(* IEC 61131-3 sources: 2026_Projet_YGO_ExcavatriceDragage/TOOLS/TEST_AUTO_CI/RESULTS/MAIN, 5 files *)

(* ---- FB_Main_EndToEnd.st ---- *)
(* =======================================================================
   🏰 FB_Main_EndToEnd : Mégabloc Machine d'Intégration Globale
   ───────────────────────────────────────────────────────────────
   🎯 Rôle : Instancie et chaîne en boucle fermée les 6 programmes de l'automate :
             PRG_02 (Acquisition) -> PRG_03 (Modes & Cycle) -> PRG_04 (Treuils/Benne)
             -> PRG_05 (Translation) -> PRG_06 (Outputs) -> PRG_07 (Supervision).
   🔄 Intègre également le rebouclage physique vers PRG_02 (SimBench).
   ======================================================================= *)

FUNCTION_BLOCK PUBLIC FB_Main_EndToEnd
VAR_INPUT
    // === 🕹️ Entrées Physiques Opérateur & Machine ===
    JoyRawX                 : INT := 0;
    JoyRawY                 : INT := 0;
    JoyDeadmanBtn           : BOOL := FALSE;
    BtnResetMachine         : BOOL := FALSE;

    // Commandes Modes IHM
    CmdMode                 : E_Mode := E_Mode.MAINT_N1;
    CmdWinchSelect          : INT := 0; // 0=Couplé, 1=M1, 2=M2

    // Conditions de Sécurité Châssis / Puissance
    EmergencyChainClosed    : BOOL := TRUE;
    PowerContactorEngaged   : BOOL := TRUE;

    // Capteurs Machine Réels
    M1_CablePosM            : REAL := 5.0;
    M2_CablePosM            : REAL := 5.0;
    M1_EncoderFault         : BOOL := FALSE;
    M2_EncoderFault         : BOOL := FALSE;
    PhaseRotationOk         : BOOL := TRUE;
END_VAR

VAR_OUTPUT
    // === 🚌 Bus Publics Inter-PRG Produits ===
    BusAcq                  : ST_AcquisitionInterPrg;
    BusModes                : ST_Modes_Autorisations;
    BusWinch                : ST_WinchInterPrg;
    BusTranslation          : ST_TranslationInterPrg;
    BusOutputs              : ST_OutputsInterPrg;
    BusBanner               : ST_HmiBanner;
END_VAR

VAR
    // Harnais des 6 sous-programmes
    prg02                   : FB_TestHarness_PRG_02;
    prg03                   : FB_TestHarness_PRG_03;
    prg04                   : FB_TestHarness_PRG_04;
    prg05                   : FB_TestHarness_PRG_05;
    prg06                   : FB_TestHarness_PRG_06;
    prg07                   : FB_TestHarness_PRG_07;
END_VAR

{region "Exécution séquentielle cyclique du Mégabloc Machine"}

// ── 1. PRG_02 : Acquisition des entrées et qualification joystick ──
prg02(
    JoyRawX                 := JoyRawX,
    JoyRawY                 := JoyRawY,
    JoyBtnRaw               := JoyDeadmanBtn,
    PowerContactorEngaged   := PowerContactorEngaged,
    EmergencyChainClosed    := EmergencyChainClosed
);
BusAcq := prg02.Data;

// ── 2. PRG_03 : Arbitrage des Modes et Séquenceur de Cycle ──
prg03(
    SelMode                 := CmdMode,
    SelJoystickWinch        := CmdWinchSelect,
    PowerContactorEngaged   := PowerContactorEngaged,
    DeadmanArmed            := BusAcq.JoystickDeadmanArmed,
    JoystickDeflected       := NOT BusAcq.JoystickYNeutral,
    BtnModeReset            := BtnResetMachine
);
BusModes := prg03.Auth;

// ── 3. PRG_04 : Contrôle Treuils M1 / M2 et Benne ──
prg04(
    AcqData                 := BusAcq,
    ModesAuth               := BusModes,
    PowerContactorEngaged   := PowerContactorEngaged,
    EmergencyChainClosed    := EmergencyChainClosed,
    M1_ContactorsReleased   := TRUE,
    M1_BrakeFeedbackOpen    := FALSE,
    M2_ContactorsReleased   := TRUE,
    M2_BrakeFeedbackOpen    := FALSE,
    BtnWinchM1Up            := FALSE,
    BtnWinchM1Down          := FALSE,
    BtnReset                := BtnResetMachine
);
BusWinch := prg04.Data;

// ── 4. PRG_05 : Contrôle Translation M3 ──
prg05(
    AcqData                 := BusAcq,
    ModesAuth               := BusModes,
    WinchM1CablePosM        := BusAcq.CablePosM1,
    WinchM2CablePosM        := BusAcq.CablePosM2,
    PowerContactorEngaged   := PowerContactorEngaged,
    EmergencyChainClosed    := EmergencyChainClosed,
    BrakeFeedbackOpen       := FALSE,
    DriveOnline             := TRUE,
    DriveOperational        := TRUE,
    BtnReset                := BtnResetMachine,
    BtnTranslationFwd       := FALSE,
    BtnTranslationRev       := FALSE
);
BusTranslation := prg05.Data;

// ── 5. PRG_06 : Barrières Finales et Génération des Sorties ──
prg06(
    WinchData               := BusWinch,
    TranslationData         := BusTranslation,
    FaultReset              := BtnResetMachine
);
BusOutputs := prg06.Data;

// ── 6. PRG_07 : Supervision et Formatage du Bandeau IHM ──
prg07(
    AcqData                 := BusAcq,
    ModesAuth               := BusModes,
    WinchData               := BusWinch,
    TranslationData         := BusTranslation,
    EmergencyChainClosed    := EmergencyChainClosed,
    PowerContactorEngaged   := PowerContactorEngaged,
    PowerCutOffActive       := FALSE,
    BtnResetMachine         := BtnResetMachine
);
BusBanner := prg07.Banner;

{endregion}
END_FUNCTION_BLOCK

(* ---- FB_TestHarness_PRG_02.st ---- *)
(* =======================================================================
   🧱 FB_TestHarness_PRG_02 : Banc d'essai unitaire pour PRG_02_Acquisition
   ───────────────────────────────────────────────────────────────
   🎯 Rôle : Isole PRG_02, injecte les entrées brutes physiques/simulation,
             exécute le bloc et expose les flux de données sortants du bus Data.
   ======================================================================= *)

FUNCTION_BLOCK PUBLIC FB_TestHarness_PRG_02
VAR_INPUT
    // === 🕹️ Entrées Joystick Brutes ===
    JoyRawX               : INT := 5000;
    JoyRawY               : INT := 5000;
    JoyBtnRaw             : BOOL;

    // === 🪝 Entrées Codeurs Brutes ===
    COD1_PosValue         : UDINT := 1000000;
    COD2_PosValue         : UDINT := 1000000;

    // === ↔️ Capteurs Translation M3 ===
    M3_PosTremie_DI       : BOOL;
    M3_PosPV_DI           : BOOL;
    M3_PosPVP2_DI         : BOOL;
    M3_PosP1_DI           : BOOL;
    M3_PosMaintenance_DI  : BOOL;

    // === 🛡️ Sécurités / Machine ===
    PowerContactorEngaged : BOOL := TRUE;
    EmergencyChainClosed  : BOOL := TRUE;

    // === 🔌 Diagnostics Réseau Simulés ===
    CanBusOperational     : BOOL := TRUE;
    JoyOperational        : BOOL := TRUE;
    EcatOperational       : BOOL := TRUE;

    // === 🧪 Commande Simulation ===
    SimulationModeActive  : BOOL := FALSE;
END_VAR

VAR_OUTPUT
    // === 🚌 Bus de données produit vers PRG_03/04/05/06/07 ===
    Data                  : ST_AcquisitionInterPrg;

    // === 🖼️ Image Qualifiée HwIn ===
    HwIn                  : ST_HardwareImage;
END_VAR

VAR
    instJoystick          : FB_Joystick;
    instDiagCanOpen       : FB_Diag_CanOpen;
    instDiagEthercat      : FB_Diag_Ethercat;
    instEncoderM1         : FB_Encoder;
    instEncoderM2         : FB_Encoder;
    instPosDecoderM3      : FB_Translation_PositionDecoder;

    diagCanDev            : ST_Diag_Device;
    diagEcatDev           : ST_Diag_Device;
    calibM1               : ST_Encoder_Calib;
    calibM2               : ST_Encoder_Calib;
    hwM1                  : ST_EncoderHw;
    hwM2                  : ST_EncoderHw;
    nxMem                 : INT := 5000;
    nyMem                 : INT := 5000;
END_VAR

{region "Corps d'exécution PRG_02 encapsulé"}
// 1. Diagnostics Réseau
diagCanDev.Online := CanBusOperational;
diagCanDev.Operational := CanBusOperational AND JoyOperational;
IF diagCanDev.Operational THEN
    diagCanDev.State := E_Diag_State.READY;
ELSE
    diagCanDev.State := E_Diag_State.INIT;
END_IF;

diagEcatDev.Online := EcatOperational;
diagEcatDev.Operational := EcatOperational;
IF diagEcatDev.Operational THEN
    diagEcatDev.State := E_Diag_State.READY;
ELSE
    diagEcatDev.State := E_Diag_State.INIT;
END_IF;

// 2. Traitement Joystick
instJoystick(
    Enable := TRUE,
    Reset := FALSE,
    ArmingPermit := TRUE,
    BusCanOpenOp := diagCanDev,
    JoystickOp := diagCanDev,
    RawX := JoyRawX,
    RawY := JoyRawY,
    RawButton := JoyBtnRaw,
    NeutralHoldTime := T#50ms,
    DeadmanArmHoldTime := T#50ms,
    DeadmanArmGraceTime := T#3s,
    DeadbandRaw := 300,
    NeutralXMem := nxMem,
    NeutralYMem := nyMem
);

Data.JoystickDeadmanArmed := instJoystick.DeadmanArmed;
Data.JoystickXNeutral     := instJoystick.AxisCmdX.AtNeutral;
Data.JoystickYNeutral     := instJoystick.AxisCmdY.AtNeutral;
Data.JoystickDirectionX   := instJoystick.DirectionX;
Data.JoystickSpeedPctX    := instJoystick.AxisCmdX.SpeedRef;

// 3. Traitement Codeurs Treuils M1 / M2
hwM1.RawPosIn := COD1_PosValue;
hwM1.SlaveOperational := EcatOperational;
instEncoderM1(
    Enable := TRUE,
    Reset := FALSE,
    HomingPermit := TRUE,
    TopPositionSensor := FALSE,
    Hw := hwM1,
    PointsPerRev := 8192,
    CableM_PerRev := 2.0,
    BypassGlobal := FALSE,
    Calib := calibM1
);
Data.CablePosM1            := instEncoderM1.Measurement.CablePosM;
Data.M1_Speed_Mps          := instEncoderM1.Measurement.Speed_Mps;
Data.M1_SignedSpeed_Mps    := instEncoderM1.Measurement.SignedSpeed_Mps;
Data.M1_SpeedValid         := instEncoderM1.Measurement.SpeedValid;
Data.M1_EncoderIncoherent  := instEncoderM1.Measurement.EncoderIncoherent;
Data.M1_EncoderFault       := instEncoderM1.EncoderFault;
Data.M1_HomedAndReliable   := instEncoderM1.HomedAndReliable;

hwM2.RawPosIn := COD2_PosValue;
hwM2.SlaveOperational := EcatOperational;
instEncoderM2(
    Enable := TRUE,
    Reset := FALSE,
    HomingPermit := TRUE,
    TopPositionSensor := FALSE,
    Hw := hwM2,
    PointsPerRev := 8192,
    CableM_PerRev := 2.0,
    BypassGlobal := FALSE,
    Calib := calibM2
);
Data.CablePosM2            := instEncoderM2.Measurement.CablePosM;
Data.M2_Speed_Mps          := instEncoderM2.Measurement.Speed_Mps;
Data.M2_SignedSpeed_Mps    := instEncoderM2.Measurement.SignedSpeed_Mps;
Data.M2_SpeedValid         := instEncoderM2.Measurement.SpeedValid;
Data.M2_EncoderIncoherent  := instEncoderM2.Measurement.EncoderIncoherent;
Data.M2_EncoderFault       := instEncoderM2.EncoderFault;
Data.M2_HomedAndReliable   := instEncoderM2.HomedAndReliable;

// 4. Décodage Position Translation M3
instPosDecoderM3(
    SensorTremie := M3_PosTremie_DI,
    SensorPV := M3_PosPV_DI,
    SensorP2 := M3_PosPVP2_DI,
    SensorP1 := M3_PosP1_DI,
    SensorMaintenance := M3_PosMaintenance_DI
);
Data.TranslationPosTremie      := instPosDecoderM3.TranslationPosTremie;
Data.TranslationPosPV          := instPosDecoderM3.TranslationPosPV;
Data.TranslationPosP2          := instPosDecoderM3.TranslationPosP2;
Data.TranslationPosP1          := instPosDecoderM3.TranslationPosP1;
Data.TranslationPosMaintenance := instPosDecoderM3.TranslationPosMaintenance;
Data.TranslationAtTremie       := instPosDecoderM3.TranslationAtTremie;
Data.TranslationAtPV           := instPosDecoderM3.TranslationAtPV;
Data.TranslationAtP2           := instPosDecoderM3.TranslationAtP2;
Data.TranslationAtP1           := instPosDecoderM3.TranslationAtP1;
Data.TranslationAtMaintenance  := instPosDecoderM3.TranslationAtMaintenance;
Data.M3_LimitSwitchFwd         := instPosDecoderM3.LimitSwitchFwd;
Data.M3_LimitSwitchRev         := instPosDecoderM3.LimitSwitchRev;
Data.M3_SensorWordIncoherent   := instPosDecoderM3.Incoherent;

// Diagnostics Cartes DI
Data.LocalDigitalIoOk := TRUE;
Data.Vh0800EndOk      := TRUE;
Data.Vh0808EtpOk      := TRUE;
Data.InputModuleFault := FALSE;
{endregion}
END_FUNCTION_BLOCK

(* ---- FB_TestHarness_PRG_03.st ---- *)
(* =======================================================================
   🧱 FB_TestHarness_PRG_03 : Banc d'essai unitaire pour PRG_03_Modes_Cycle
   ───────────────────────────────────────────────────────────────
   🎯 Rôle : Isole PRG_03, injecte les sélections de modes et commandes cycle,
             exécute FB_Modes et FB_Cycle, et expose le bus ST_Modes_Autorisations.
   ======================================================================= *)

FUNCTION_BLOCK PUBLIC FB_TestHarness_PRG_03
VAR_INPUT
    // === 🎚️ Sélections IHM Modes ===
    SelMode                 : E_Mode := E_Mode.MAINT_N1;
    BtnModeReset            : BOOL;
    SelSyncEnable           : BOOL := TRUE;
    InhibitM1Request        : BOOL := FALSE;
    InhibitM2Request        : BOOL := FALSE;
    SelHomingApproachEnable : BOOL := FALSE;
    SelJoystickWinch        : INT := 1; // 1 = M1, 2 = M2, 0 = Both
    TglMaintenanceZoneAccess: BOOL := FALSE;

    // === 🛡️ Sécurités Machine ===
    PowerContactorEngaged   : BOOL := TRUE;
    EncoderFaultPresent     : BOOL := FALSE;

    // === 🔄 Commandes Cycle Semi-Auto ===
    BtnStartCycle           : BOOL;
    BtnAbortCycle           : BOOL;
    BtnCycleReset           : BOOL;
    DeadmanArmed            : BOOL := TRUE;
    JoystickDeflected       : BOOL := TRUE;
    HeartbeatIhmOk          : BOOL := TRUE;

    // === 📏 Données mesurées / retours treuils ===
    M1_CablePosM            : REAL := 5.0;
    M2_CablePosM            : REAL := 5.0;
    M1_SpeedMps             : REAL := 0.0;
    M2_SpeedMps             : REAL := 0.0;
    Benne_IsClosed          : BOOL := TRUE;
    Benne_IsOpen            : BOOL := FALSE;
    Benne_IsRoughlyClosed   : BOOL := TRUE;
    HomedM1                 : BOOL := TRUE;
    HomedM2                 : BOOL := TRUE;
END_VAR

VAR_OUTPUT
    // === 🎚️ Bus d'Autorisations Produit vers PRG_04/05/06/07 ===
    Auth                    : ST_Modes_Autorisations;

    // === 🔄 Séquenceur de Cycle Semi-Auto ===
    CycleStep               : E_CycleStep;
    CycleBusy               : BOOL;
    CycleDone               : BOOL;
    CycleError              : BOOL;
    CycleStateStr           : STRING(80);
END_VAR

VAR
    instModes               : FB_Modes;
    instCycleSemiAuto       : FB_Cycle;
    countMem                : INT := 0;
END_VAR

{region "Corps d'exécution PRG_03 encapsulé"}
// 1. Arbitrage des Modes Machine
instModes(
    Enable                  := TRUE,
    Reset                   := BtnModeReset,
    PowerContactorEngaged   := PowerContactorEngaged,
    SelMode                 := SelMode,
    SelSyncEnable           := SelSyncEnable,
    InhibitM1Request        := InhibitM1Request,
    InhibitM2Request        := InhibitM2Request,
    SelHomingApproachEnable := SelHomingApproachEnable,
    EncoderFaultPresent     := EncoderFaultPresent,
    JoystickWinchSelectRequest := SelJoystickWinch,
    SelMaintenanceZoneAccess := TglMaintenanceZoneAccess
);

Auth := instModes.Auth;

// 2. Séquenceur de Cycle Semi-Automatique
instCycleSemiAuto(
    Enable                  := (Auth.Mode = E_Mode.SEMI_AUTO),
    Reset                   := BtnCycleReset,
    PowerContactorEngaged   := PowerContactorEngaged,
    Mode                    := Auth.Mode,
    CycleMotionPermit       := JoystickDeflected,
    DeadmanArmed            := DeadmanArmed,
    HeartbeatIhmOk          := HeartbeatIhmOk,
    StartCycle              := BtnStartCycle,
    AbortCycle              := BtnAbortCycle,
    SelTarget               := 1,
    SetDepthM               := -12.0,
    SetOffsetM              := 1.5,
    KoboldContactFond       := FALSE,
    LimitLegalReached       := FALSE,
    LimitLegalDepthM        := -15.0,
    WinchSyncError          := FALSE,
    WinchSyncDeltaM         := 0.0,
    M1_CablePosM            := M1_CablePosM,
    M2_CablePosM            := M2_CablePosM,
    M1_MeasuredSpeedMps     := M1_SpeedMps,
    M2_MeasuredSpeedMps     := M2_SpeedMps,
    SpeedMismatchThresholdMps := 1.5,
    SpeedMismatchTimeout    := T#500ms,
    CableLimitM1AscentM     := 7.5,
    Translation_At_P1       := FALSE,
    Translation_At_Tremie   := TRUE,
    Translation_At_Maintenance := FALSE,
    Translation_Busy        := FALSE,
    Translation_Done        := TRUE,
    Benne_Busy              := FALSE,
    Benne_Done              := TRUE,
    Benne_IsOpen            := Benne_IsOpen,
    Benne_IsClosed          := Benne_IsClosed,
    Benne_IsRoughlyClosed   := Benne_IsRoughlyClosed,
    HomedM1                 := HomedM1,
    HomedM2                 := HomedM2,
    TopPositionSensor       := FALSE,
    HomingRequest           := FALSE,
    SampleCount             := countMem
);

CycleStep     := instCycleSemiAuto.CycleStep;
CycleBusy     := instCycleSemiAuto.Busy;
CycleDone     := instCycleSemiAuto.Done;
CycleError    := instCycleSemiAuto.Error;
CycleStateStr := instCycleSemiAuto.CycleStateStr;

{endregion}
END_FUNCTION_BLOCK

(* ---- FB_TestHarness_PRG_04.st ---- *)
(* =======================================================================
   🧱 FB_TestHarness_PRG_04 : Banc d'essai unitaire pour PRG_04_Treuils_Benne
   ───────────────────────────────────────────────────────────────
   🎯 Rôle : Isole PRG_04, consomme les bus de données de PRG_02 (Joystick,
             mesures câbles) et PRG_03 (Modes/Autorisations), exécute
             les treuils M1/M2, sécurités, synchro et benne, et publie ST_WinchInterPrg.
   ======================================================================= *)

FUNCTION_BLOCK PUBLIC FB_TestHarness_PRG_04
VAR_INPUT
    // === 📥 Bus d'Entrée issus de PRG_02 (Acquisition) ===
    AcqData                 : ST_AcquisitionInterPrg;

    // === 📥 Bus d'Entrée issus de PRG_03 (Modes) ===
    ModesAuth               : ST_Modes_Autorisations;

    // === 🛡️ Sécurités & Hardware Machine ===
    PowerContactorEngaged   : BOOL := TRUE;
    EmergencyChainClosed    : BOOL := TRUE;
    M1_ContactorsReleased   : BOOL := TRUE;
    M2_ContactorsReleased   : BOOL := TRUE;
    M1_BrakeFeedbackOpen    : BOOL := FALSE;
    M2_BrakeFeedbackOpen    : BOOL := FALSE;

    // === 🎛️ Commandes IHM Directes ===
    BtnReset                : BOOL := FALSE;
    BtnBucketOpen           : BOOL := FALSE;
    BtnBucketClose          : BOOL := FALSE;
    BtnWinchM1Up            : BOOL := FALSE;
    BtnWinchM1Down          : BOOL := FALSE;
END_VAR

VAR_OUTPUT
    // === 🚌 Bus Inter-PRG produit vers PRG_02/03/06/07 ===
    Data                    : ST_WinchInterPrg;
END_VAR

VAR
    instWinchSync           : FB_WinchSync;
    instBucket              : FB_Bucket;
    instSafetyWinchM1       : FB_Safety_Winch;
    instSafetyWinchM2       : FB_Safety_Winch;
    instWinchM1             : FB_Winch;
    instWinchM2             : FB_Winch;

    speedCfg                : ST_WinchSpeedConfig;
    bucketCfg               : ST_BucketConfig;
    m1StartStop             : BOOL;
    m1Direction             : INT;
    m1SpeedRef              : REAL;
    stepTable               : ST_SpeedStepTable;
END_VAR

{region "Corps d'exécution PRG_04 encapsulé"}
// 1. Initialisation configurations de référence
stepTable.StepThreshold_Pct[1] := 10.0;
stepTable.StepThreshold_Pct[2] := 30.0;
stepTable.StepThreshold_Pct[3] := 50.0;
stepTable.StepThreshold_Pct[4] := 70.0;
stepTable.StepThreshold_Pct[5] := 90.0;
stepTable.P1R1 := TRUE;
stepTable.P2R1 := TRUE;
stepTable.P3R1 := TRUE;
stepTable.P4R1 := TRUE;
stepTable.P5R1 := TRUE;
bucketCfg.OffsetOpenM := 0.0;
bucketCfg.OffsetCloseM := 15.0;
bucketCfg.CoherenceLimitM := 1.0;

// 2. Sécurités Treuil M1
instSafetyWinchM1(
    Enable                  := (ModesAuth.Mode = E_Mode.MAINT_N1 OR ModesAuth.Mode = E_Mode.MAINT_N2 OR ModesAuth.Mode = E_Mode.SEMI_AUTO),
    Reset                   := BtnReset,
    Mode                    := ModesAuth.Mode,
    PowerContactorEngaged   := PowerContactorEngaged,
    JoystickOnline          := TRUE,
    JoystickOperational     := TRUE,
    HeartbeatIhmOk          := TRUE,
    EncoderAvailable        := NOT AcqData.M1_EncoderFault,
    ThermalFeedback         := FALSE,
    BrakeThermalFeedback    := FALSE,
    SlackCableDetected      := FALSE,
    PhaseRotationOk         := TRUE,
    TopPositionSensor       := TRUE,

    FwdRevSpeedFeedbackOff  := M1_ContactorsReleased,
    BrakeFeedback           := M1_BrakeFeedbackOpen,
    JoystickYNeutral        := AcqData.JoystickYNeutral,
    CablePosM               := AcqData.CablePosM1,
    CfgCableLimitDescentM   := -20.0,
    TopLimitM               := 7.5,
    MeasuredSpeedMps        := AcqData.M1_Speed_Mps,
    MeasuredSpeedSignedMps  := AcqData.M1_SignedSpeed_Mps,
    MeasuredSpeedValid      := AcqData.M1_SpeedValid
);
Data.WinchM1Safety.SafeStop      := instSafetyWinchM1.SafeStop;
Data.WinchM1Safety.DescendPermit := instSafetyWinchM1.DescendPermit;
Data.WinchM1Safety.AscentPermit  := instSafetyWinchM1.AscentPermit;
Data.WinchM1Safety.PowerCutOff   := instSafetyWinchM1.PowerCutOff;

// 3. Sécurités Treuil M2
instSafetyWinchM2(
    Enable                  := (ModesAuth.Mode = E_Mode.MAINT_N1 OR ModesAuth.Mode = E_Mode.MAINT_N2 OR ModesAuth.Mode = E_Mode.SEMI_AUTO),
    Reset                   := BtnReset,
    Mode                    := ModesAuth.Mode,
    PowerContactorEngaged   := PowerContactorEngaged,
    JoystickOnline          := TRUE,
    JoystickOperational     := TRUE,
    HeartbeatIhmOk          := TRUE,
    EncoderAvailable        := NOT AcqData.M2_EncoderFault,
    ThermalFeedback         := FALSE,
    BrakeThermalFeedback    := FALSE,
    SlackCableDetected      := FALSE,

    PhaseRotationOk         := TRUE,
    TopPositionSensor       := TRUE,
    FwdRevSpeedFeedbackOff  := M2_ContactorsReleased,

    BrakeFeedback           := M2_BrakeFeedbackOpen,
    JoystickYNeutral        := AcqData.JoystickYNeutral,
    CablePosM               := AcqData.CablePosM2,
    CfgCableLimitDescentM   := -20.0,
    TopLimitM               := 7.5,
    MeasuredSpeedMps        := AcqData.M2_Speed_Mps,
    MeasuredSpeedSignedMps  := AcqData.M2_SignedSpeed_Mps,
    MeasuredSpeedValid      := AcqData.M2_SpeedValid
);
Data.WinchM2Safety.SafeStop      := instSafetyWinchM2.SafeStop;
Data.WinchM2Safety.DescendPermit := instSafetyWinchM2.DescendPermit;
Data.WinchM2Safety.AscentPermit  := instSafetyWinchM2.AscentPermit;
Data.WinchM2Safety.PowerCutOff   := instSafetyWinchM2.PowerCutOff;

// 4. Commande Treuil M1 (arbitrage Joystick + Boutons)
m1StartStop := (AcqData.JoystickDeadmanArmed AND (AcqData.JoystickDirectionX = 0) AND NOT AcqData.JoystickYNeutral AND (ModesAuth.JoystickWinchSelectArbitrated = 1 OR ModesAuth.JoystickWinchSelectArbitrated = 0))
               OR BtnWinchM1Up OR BtnWinchM1Down;

IF BtnWinchM1Up THEN
    m1Direction := 1;
    m1SpeedRef  := 50.0;
ELSIF BtnWinchM1Down THEN
    m1Direction := -1;
    m1SpeedRef  := 50.0;
ELSIF AcqData.JoystickDeadmanArmed AND NOT AcqData.JoystickYNeutral THEN
    m1Direction := 1; // Commande de montée treuil M1
    m1SpeedRef  := 60.0;

ELSE
    m1Direction := 0;
    m1SpeedRef  := 0.0;
END_IF;

instWinchM1(
    Enable                  := (ModesAuth.Mode = E_Mode.MAINT_N1 OR ModesAuth.Mode = E_Mode.MAINT_N2 OR ModesAuth.Mode = E_Mode.SEMI_AUTO),
    Reset                   := BtnReset,
    PowerContactorEngaged   := PowerContactorEngaged,
    SafeStop                := Data.WinchM1Safety.SafeStop,
    StartStop               := m1StartStop,
    Direction               := m1Direction,
    SpeedRefPct             := m1SpeedRef,
    Mode                    := ModesAuth.Mode,
    DescendPermit           := Data.WinchM1Safety.DescendPermit,
    AscentPermit            := Data.WinchM1Safety.AscentPermit,
    CablePosM               := AcqData.CablePosM1,
    Homed                   := TRUE,
    MaxStepAscent           := 5,
    CfgMaxStepDescente      := 3,
    SpeedStepTable          := stepTable,
    FwdRevSpeedFeedbackOff  := M1_ContactorsReleased
);

// Remplissage bus de sortie Data
Data.WinchM1FinalInterlockRequest.RequestedRelayFwd          := instWinchM1.RelayFwd;
Data.WinchM1FinalInterlockRequest.RequestedRelayRev          := instWinchM1.RelayRev;
Data.WinchM1FinalInterlockRequest.RequestedContactor1        := instWinchM1.Contactor1;
Data.WinchM1FinalInterlockRequest.RequestedContactor2        := instWinchM1.Contactor2;
Data.WinchM1FinalInterlockRequest.RequestedContactor3        := instWinchM1.Contactor3;
Data.WinchM1FinalInterlockRequest.RequestedContactor4        := instWinchM1.Contactor4;
Data.WinchM1FinalInterlockRequest.RequestedStep              := instWinchM1.StepNumber;
Data.WinchM1FinalInterlockRequest.PowerCutOff               := Data.WinchM1Safety.PowerCutOff;
Data.WinchM1FinalInterlockRequest.SafeStop                  := Data.WinchM1Safety.SafeStop;

Data.M1LogicRequestSpeedRef_Pct                             := m1SpeedRef;
Data.WinchM1State.StepNumber                                := instWinchM1.StepNumber;
Data.WinchM1State.RelayFwd                                  := instWinchM1.RelayFwd;
Data.WinchM1State.RelayRev                                  := instWinchM1.RelayRev;
{endregion}
END_FUNCTION_BLOCK

(* ---- FB_TestHarness_PRG_05.st ---- *)
(* =======================================================================
   🧱 FB_TestHarness_PRG_05 : Banc d'essai unitaire pour PRG_05_Translation
   ───────────────────────────────────────────────────────────────
   🎯 Rôle : Isole PRG_05, consomme les bus de données de PRG_02 (Position,
             capteurs, joystick X), PRG_03 (Modes/Autorisations) et PRG_04 (Hauteur treuils),
             exécute FB_Translation et FB_Safety_Translation, et publie ST_TranslationInterPrg.
   ======================================================================= *)

FUNCTION_BLOCK PUBLIC FB_TestHarness_PRG_05
VAR_INPUT
    // === 📥 Bus d'Entrée issus de PRG_02 (Acquisition) ===
    AcqData                 : ST_AcquisitionInterPrg;

    // === 📥 Bus d'Entrée issus de PRG_03 (Modes) ===
    ModesAuth               : ST_Modes_Autorisations;

    // === 📥 Bus d'Entrée issus de PRG_04 (Treuils / Hauteur câble) ===
    WinchM1CablePosM        : REAL := 5.0;
    WinchM2CablePosM        : REAL := 5.0;

    // === 🛡️ Sécurités & Hardware Machine ===
    PowerContactorEngaged   : BOOL := TRUE;
    EmergencyChainClosed    : BOOL := TRUE;
    BrakeFeedbackOpen       : BOOL := FALSE;
    DriveOnline             : BOOL := TRUE;
    DriveOperational        : BOOL := TRUE;

    // === 🎛️ Commandes IHM Directes ===
    BtnReset                : BOOL := FALSE;
    BtnTranslationFwd       : BOOL := FALSE;
    BtnTranslationRev       : BOOL := FALSE;
END_VAR

VAR_OUTPUT
    // === 🚌 Bus Inter-PRG produit vers PRG_03/06/07 ===
    Data                    : ST_TranslationInterPrg;
END_VAR

VAR
    instTranslationM3       : FB_Translation;
    instSafetyTranslationM3 : FB_Safety_Translation;

    m3StartStop             : BOOL;
    m3Direction             : INT;
    m3SpeedRef              : REAL;
    m3HeightOk              : BOOL;
END_VAR

{region "Corps d'exécution PRG_05 encapsulé"}
// 1. Interlock Hauteur Treuils (Treuils doivent être au-dessus du seuil mini pour translater)
m3HeightOk := (WinchM1CablePosM >= 2.0) AND (WinchM2CablePosM >= 2.0);

// 2. Sécurité Translation M3
instSafetyTranslationM3(
    Enable                  := (ModesAuth.Mode = E_Mode.MAINT_N1 OR ModesAuth.Mode = E_Mode.MAINT_N2 OR ModesAuth.Mode = E_Mode.SEMI_AUTO),
    Reset                   := BtnReset,
    PowerContactorEngaged   := PowerContactorEngaged,
    Mode                    := ModesAuth.Mode,
    JoystickOnline          := TRUE,
    JoystickOperational     := TRUE,
    HeartbeatIhmOk          := TRUE,
    PhaseRotationOk         := TRUE,
    BrakeThermalFeedback    := FALSE,
    DriveOnline             := DriveOnline,
    DriveOperational        := DriveOperational,
    DriveStatusWord         := 16#0000,
    DriveActualFreqHz       := 0.0,
    BrakeFeedback           := BrakeFeedbackOpen,
    BrakeCmd                := FALSE,
    Direction               := m3Direction,
    LimitSwitchFwd          := AcqData.M3_LimitSwitchFwd,
    LimitSwitchRev          := AcqData.M3_LimitSwitchRev,
    SensorWordIncoherent    := AcqData.M3_SensorWordIncoherent
);

Data.TranslationSafety.SafeStop    := instSafetyTranslationM3.SafeStop;
Data.TranslationSafety.PowerCutOff := instSafetyTranslationM3.PowerCutOff;

// 3. Arbitrage Commande Translation (Joystick X ou Boutons)
m3StartStop := (AcqData.JoystickDeadmanArmed AND (AcqData.JoystickDirectionX <> 0) AND m3HeightOk)
               OR BtnTranslationFwd OR BtnTranslationRev;

IF BtnTranslationFwd THEN
    m3Direction := 1;
    m3SpeedRef  := 50.0;
ELSIF BtnTranslationRev THEN
    m3Direction := -1;
    m3SpeedRef  := 50.0;
ELSIF AcqData.JoystickDeadmanArmed AND (AcqData.JoystickDirectionX <> 0) AND m3HeightOk THEN
    m3Direction := AcqData.JoystickDirectionX;
    m3SpeedRef  := AcqData.JoystickSpeedPctX;
ELSE
    m3Direction := 0;
    m3SpeedRef  := 0.0;
END_IF;

// 4. Pilotage M3
instTranslationM3(
    Enable                  := (ModesAuth.Mode = E_Mode.MAINT_N1 OR ModesAuth.Mode = E_Mode.MAINT_N2 OR ModesAuth.Mode = E_Mode.SEMI_AUTO),
    Reset                   := BtnReset,
    PowerContactorEngaged   := PowerContactorEngaged,
    Mode                    := ModesAuth.Mode,
    StartStop               := m3StartStop,
    SafeStop                := Data.TranslationSafety.SafeStop,
    Direction               := m3Direction,
    SpeedRefPct             := m3SpeedRef,
    PositionSensorTarget    := FALSE,
    SlowdownSensorTremie    := AcqData.TranslationAtPV,
    SlowdownSensorMaintenance := AcqData.TranslationAtP1,
    SlowdownSensorP1        := AcqData.TranslationAtP2,
    LimitSwitchFwd          := AcqData.M3_LimitSwitchFwd,
    LimitSwitchRev          := AcqData.M3_LimitSwitchRev,
    DriveStatusWord         := 16#0081,
    DriveActualFreqHz       := 0.0,
    BrakeFeedback           := BrakeFeedbackOpen,
    BrakeDelayContactClose  := T#0ms,
    BrakeDelayMagnetise     := T#0ms,
    CfgRampAccelRate        := 1000.0
);

// 5. Remplissage Bus Sortie Data
Data.TranslationFinalInterlockRequest.Enable                    := instTranslationM3.Enable;
Data.TranslationFinalInterlockRequest.Reset                     := BtnReset;
Data.TranslationFinalInterlockRequest.PowerContactorEngaged     := PowerContactorEngaged;
Data.TranslationFinalInterlockRequest.SafeStop                  := Data.TranslationSafety.SafeStop;
Data.TranslationFinalInterlockRequest.PowerCutOff               := Data.TranslationSafety.PowerCutOff;
Data.TranslationFinalInterlockRequest.BrakeReleaseRequest       := instTranslationM3.BrakeReleaseRequest;
Data.TranslationFinalInterlockRequest.RequestedDriveControlWord := instTranslationM3.RequestedDriveControlWord;
Data.TranslationFinalInterlockRequest.RequestedDriveFreqHz      := instTranslationM3.RequestedDriveFreqHz;

Data.TranslationState.ActiveDirection                          := m3Direction;
Data.TranslationState.ActiveSpeedRef_Pct                       := m3SpeedRef;
Data.TranslationState.Busy                                     := instTranslationM3.Status.Busy;
{endregion}
END_FUNCTION_BLOCK
